TYPE ST_TCP_Parameter :
STRUCT
	Parameter		:	INT;
	ControlWord		:	INT;
	DataType		:	INT;
	In_DataLowWord	:	WORD;
	In_DataHighWord	:	WORD;	
	Out_DataLowWord	:	WORD;
	Out_DataHighWord:	WORD;	
	
END_STRUCT
END_TYPE

(* stored: Version 1.1.0.1, ProductVersion 3.1.4024.12
   DUT ST_TCP_Parameter: Id {b95a28cc-e365-4074-b876-ce84ca76134c} *)
